{attribute 'pack_mode' := '1'}
TYPE ClearAxisFaults EXTENDS IncomingMessage :
STRUCT
	axisIndex: DINT; (* 1 or 2.*)
END_STRUCT
END_TYPE

(* stored: Version 1.1.0.1, ProductVersion 3.1.4022.12
   DUT ClearAxisFaults: Id {f831fdab-76e9-4ec8-a9c6-ad90c6b44f97} *)
